TYPE CommandBlockGeneric :
UNION
	base : CommandBlockBase;
	position : CommandBlockPos;
END_UNION
END_TYPE

(* stored: Version 1.1.0.1, ProductVersion 3.1.4020.12
   DUT CommandBlockGeneric: Id {62c6cccb-2d2a-4621-abb3-49c6aff3e548} *)
